// SIMATIC S7-200 project (STEP 7-Micro/WIN), CPU 224XP REL 02.00

SYMBOL_TABLE DR03
S1_0300_AdjDigits0 VW0      // Scale1 - Adjusting digits for zero point
S1_0302_AdjDigits1 VW2      // Scale1 - Adjusting digits for adjusting weight 1
S1_0304_AdjDigits2 VW4      // Scale1 - Adjusting digits for adjusting weight 2
S1_0306_AdjWeight1 VW6      // Scale1 - Adjusting weight 1
S1_0308_AdjWeight2 VW8      // Scale1 - Adjusting weight 2
S1_0310_CharVal  VB10     // Scale1 - Characteristic value [mV/V]
S1_0311_MeasuremTime VB11     // Scale1 - Measurement time, 0=20ms, 1=33,33ms
S1_0312_LimFrequ VB12     // Scale1 - Limit frequency for low pass filter fg
S1_0313_DepthAvValFiltr VB13     // Scale1 - Depth of average value filter [0..255]
S1_0314_ScaleName_maxL VB14     // Scale1 - Scale name, max. length (bytes)
S1_0315_ScaleName_strg VB15     // Scale1 - Scale name, STRING[10]
S1_0326_MinWeight VW26     // Scale1 - Minimum weight for weighing range
S1_0328_MaxWeight VW28     // Scale1 - Maximum weight for weighing range
S1_0330_NumeralStep VW30     // Scale1 - Numeral step (1, 2, 5, 10, 20)
S1_0332_StandstillRange VW32     // Scale1 - Standstill range in weight unit
S1_0334_StandstillTime VD34     // Scale1 - Standstill time in ms
S1_0338_DecimalPoint VB38     // Scale1 - Decimal place for remote display and       ASCII weight output (0...5)
S1_0339_NegZeroRange VB39     // Scale1 - Negative range of zero setting device                   [in % of WBB.]
S1_0340_PosZeroRange VB40     // Scale1 - Positive range of zero setting device                   [in % of WBB.]
S1_0341_TareMax  VB41     // Scale1 - Subtractive tare device range in % of weighing range
S1_0342_TTYinterface VW42     // Scale1 - 0: Siebert S102, 1: ASCII protocol
S1_0344_Res_maxL VB44     // Scale1 - Reserved, max. length (bytes)
S1_0345_Res_strg VB45     // Scale1 - Reserved, STRING[4]
S1_0350_Unit_maxL VB50     // Scale1 - Weight unit for display, max. length (bytes)
S1_0351_Unit_strg VB51     // Scale1 - Weight unit for display, STRING[4]
END_SYMBOL_TABLE

SYMBOL_TABLE DR04
S1_0400_SwOnWeightLim1 VW56     // Scale1 - Switch on point, limit value 1
S1_0402_SwOffWeightLim1 VW58     // Scale1 - Switch off point, limit value 1
S1_0404_SwOnWeightLim2 VW60     // Scale1 - Switch on point, limit value 2
S1_0406_SwOffWeightLim VW62     // Scale1 - Switch off point, limit value 2
S1_0408_LimValParamFlag VB64     // Scale1 - Bit0: 0=lim1 on gross, 1=lim1 on net;                Bit1: --> lim2
S1_0409_Res1     VB65     // Scale1 - Reserve 1
END_SYMBOL_TABLE

SYMBOL_TABLE DR09
S1_0900_ModuleName_maxL VB66     // Scale1 - Name of weighing module, max. length (bytes)
S1_0901_ModuleName_strg VB67     // Scale1 - Name of weighing module, STRING[10]
S1_0912_MLFB_maxL VB78     // Scale1 - MLFB order number, max. length (bytes)
S1_0913_MLFB_strg VB79     // Scale1 - MLFB order number, STRING[20]
S1_0934_Edition1HW VW100    // Scale1 - HW version
S1_0936_FWversion_maxL VB102    // Scale1 - FW version, max. length (bytes)
S1_0937_FWversion_strg VB103    // Scale1 - FW version, STRING[4]
S1_0942_CRCpackage VW108    // Scale1 - Depending on code
END_SYMBOL_TABLE

SYMBOL_TABLE DR15
S1_1500_TareInpVal VW110    // Scale1 - Tare input value (preset Tare pT)
END_SYMBOL_TABLE

SYMBOL_TABLE DR26
S1_2600_Checksum VW112    // Scale1 - Checksum
S1_2602_Res      VB114    // Scale1 - Reserved
S1_2603_PresetTare VB115    // Scale1 - 1 = Tare memory contains ext. default value
S1_2604_Tare_x100 VD116    // Scale1 - Tare weight * 100
S1_2608_ZeroSetVal_x100 VD120    // Scale1 - Zero set value * 100 (set during zero setting)
END_SYMBOL_TABLE

SYMBOL_TABLE DR30
S1_3000_Checksum VW124    // Scale1 - Checksum CRC16
S1_3002_ScaleStatus VW126    // Scale1 - Scale status
S1_3004_OpErrorBits VB128    // Scale1 - Operating error bits
S1_3005_Res1     VB129    // Scale1 - Reserve 1
S1_3006_GrossProcessVal VW130    // Scale1 - Gross weight
S1_3008_NetProcessVal VW132    // Scale1 - Net weight
S1_3010_TareProcessVal VW134    // Scale1 - Tare weight
S1_3012_GNweight VW136    // Scale1 - B/N weight value to display
S1_3014_GNweight10 VD138    // Scale1 - B/N weight value with 10x resolution (basis for ASCII weight value)
S1_3018_TareWeight VW142    // Scale1 - Tare weight value
S1_3020_UnfiltRawVal VW144    // Scale1 - Unfiltered digital value from ADU
S1_3022_FiltRawVal VW146    // Scale1 - Filtered digital value
S1_3024_WghtASCII_maxL VB148    // Scale1 - ASCII weight value, max. length (bytes)
S1_3025_WghtASCII_strg VB149    // Scale1 - ASCII weight value, STRING[14]
S1_3040_Millisecond VW164    // Scale1 - Runtime – Milliseconds (0....999)
S1_3042_Second   VB166    // Scale1 - Runtime – Seconds (0...59)
S1_3043_Minute   VB167    // Scale1 - Runtime – Minutes (0...59)
S1_3044_Hour     VW168    // Scale1 - Runtime – Hours (0...32000)
END_SYMBOL_TABLE

SYMBOL_TABLE MS
Q_S1_Actual_Process_Val VB200    // Scale1 - VBn
Q_S1_Reserve_1   VB201    // Scale1 - VBn+1
Q_S1_Process_Value VW202    // Scale1 - VWn+2
Q_S1_Bit_Messages VB204    // Scale1 - VBn+4
Q_S1_Bit_Messages_Bit0 V204.0   // Scale1 - VBn+4, Bit0, command in progress
Q_S1_Bit_Messages_Bit1 V204.1   // Scale1 - VBn+4, Bit1, command finished ok (TRUE for 1 cycle)
Q_S1_Bit_Messages_Bit2 V204.2   // Scale1 - VBn+4, Bit2, command error (synchronous error) has occurred (TRUE for 1 cycle)
Q_S1_Bit_Messages_Bit3 V204.3   // Scale1 - VBn+4, Bit3, Read/Write-Parameter-Mode is supported
Q_S1_Bit_Messages_Bit4 V204.4   // Scale1 - VBn+4, Bit4, Processvalue not valid!
Q_S1_Bit_Messages_Bit5 V204.5   // Scale1 - VBn+4, Bit5, Reserve
Q_S1_Bit_Messages_Bit6 V204.6   // Scale1 - VBn+4, Bit6, Reserve
Q_S1_Bit_Messages_Bit7 V204.7   // Scale1 - VBn+4, Bit7, Reserve
Q_S1_Sync_Error_Code VB205    // Scale1 - VBn+5
Q_S1_Async_Error_Bits VB206    // Scale1 - VBn+6
Q_S1_Async_Error_Bit0 V206.0   // Scale1 - VBn+6, Bit0, Reboot due to RAM error
Q_S1_Async_Error_Bit1 V206.1   // Scale1 - VBn+6, Bit1, Reboot due to watchdog error
Q_S1_Async_Error_Bit2 V206.2   // Scale1 - VBn+6, Bit2, 24DC power supply faulty/missing
Q_S1_Async_Error_Bit3 V206.3   // Scale1 - VBn+6, Bit3, Number overflow in weight calculation
Q_S1_Async_Error_Bit4 V206.4   // Scale1 - VBn+6, Bit4, Parameter error
Q_S1_Async_Error_Bit5 V206.5   // Scale1 - VBn+6, Bit5, AD converter at limit of measuring range
Q_S1_Async_Error_Bit6 V206.6   // Scale1 - VBn+6, Bit6, Minimum voltage understhot in sensor line
Q_S1_Async_Error_Bit7 V206.7   // Scale1 - VBn+6, Bit7, AD converter fault
Q_S1_Refresh_Counter VB207    // Scale1 - VBn+7
Q_S1_Scale_Status_Bits VW208    // Scale1 - VWn+8
Q_S1_Scale_Status_Bit0 V209.0   // Scale1 - VWn+8, Bit0, Limit value 1 has responded
Q_S1_Scale_Status_Bit1 V209.1   // Scale1 - VWn+8, Bit1, Limit value 2 has responded
Q_S1_Scale_Status_Bit2 V209.2   // Scale1 - VWn+8, Bit2, Tare memory occupied (<>0)
Q_S1_Scale_Status_Bit3 V209.3   // Scale1 - VWn+8, Bit3, Tare memory contains ext. default value
Q_S1_Scale_Status_Bit4 V209.4   // Scale1 - VWn+8, Bit4, Gross weighing range exceeded or understhot (>9 display steps)
Q_S1_Scale_Status_Bit5 V209.5   // Scale1 - VWn+8, Bit5, Gross less than ± 0.25d (d corresponds to set numeral step)
Q_S1_Scale_Status_Bit6 V209.6   // Scale1 - VWn+8, Bit6, Standstill exists
Q_S1_Scale_Status_Bit7 V209.7   // Scale1 - VWn+8, Bit7, Module calibrated
Q_S1_Scale_Status_Bit8 V208.0   // Scale1 - VWn+8, Bit8, Write protect switch active
Q_S1_Scale_Status_Bit9 V208.1   // Scale1 - VWn+8, Bit9, Min. weighing range undershot
Q_S1_Scale_Status_Bit10 V208.2   // Scale1 - VWn+8, Bit10, Reserve
Q_S1_Scale_Status_Bit11 V208.3   // Scale1 - VWn+8, Bit11, Reserve
Q_S1_Scale_Status_Bit12 V208.4   // Scale1 - VWn+8, Bit12, Reserve
Q_S1_Scale_Status_Bit13 V208.5   // Scale1 - VWn+8, Bit13, Reserve
Q_S1_Scale_Status_Bit14 V208.6   // Scale1 - VWn+8, Bit14, startup is running
Q_S1_Scale_Status_Bit15 V208.7   // Scale1 - VWn+8, Bit15, Global module fault / operating error (SF)
Q_S1_Select_Process_Val VB210    // Scale1 - VBn+10
I_S1_Command_Code VB211    // Scale1 - VBn+11
I_S1_Command_Bits VB212    // Scale1 - VBn+12
Q_S1_Reserve_2   VB213    // Scale1 - VBn+13
I_S1_Preset_Tare_Value VW214    // Scale1 - VWn+14
Q_S1_Lifebit_Counter VW216    // Scale1 - VWn+16
Q_S1_Lib_Error_Bits VW218    // Scale1 - VWn+18
Q_S1_RW_Mode_DS_Nr VB220    // Scale1 - VBn+20
Q_S1_RW_Mode_Byte_Offse VB221    // Scale1 - VBn+21
Q_S1_RW_Mode_Write_Data VW222    // Scale1 - VWn+22
Q_S1_RW_Mode_Read_Data VW224    // Scale1 - VWn+24
END_SYMBOL_TABLE

SYMBOL_TABLE User
Error_MS_add     VW298    // Error word of SBR "MicroScale_additional"
Error_Messages1  VW300    // To be displayed at the TP
Error_Messages2  VW302    // To be displayed at the TP
Error_Messages3  VW304    // To be displayed at the TP
Messages_Erase   V306.0   // Button on TP
Command_Trigger  V260.0
Busy             V260.1
Done             V260.2
Aborted          V260.3
Command_Code     VB261
DR               VB262
Offset           VB263
Length           VB264
END_SYMBOL_TABLE

SYMBOL_TABLE MS_add
_S1_Command_Code VB170    // Scale1 - VBn+11
_S1_Word_LoopCounter VB171
_S1_Offset       VB172
_S1_Bit_Messages VB173    // Scale1 - Bit-Messages (Siwarex => PLC)
_S1_Command_INPR V173.0   // Scale1 - command in progress
_S1_Command_FOK  V173.1   // Scale1 - command finished ok
_S1_Command_ERR  V173.2   // Scale1 - command error has occurred
_S1_DR_supported V173.3   // Scale1 - SIWAREX Module supports data record transfer
_S1_Result_bits  VB174
_S1_Busy         V174.0   // Scale1 - identic to OUT parameter
_S1_Done         V174.1
_S1_Aborted      V174.2
_S1_Bytetransfer V174.3
_S1_Err          V174.4
_S1_SequStates   VW175    // Scale1 - Sequencer states
_S1_SequState_08 V176.0   // Scale1 - Waiting for Command_FOK/_ERR of cmd 205
_S1_SequState_09 V176.1   // Scale1 - not used
_S1_SequState_10 V176.2   // Scale1 - Waiting for Actual_Process_Value = prev. Value
_S1_SequState_11 V176.3   // Scale1 - Waiting for next cycle
_S1_SequState_12 V176.4   // Scale1 - Waiting for Actual_Process_Value = 7
_S1_SequState_13 V176.5
_S1_SequState_14 V176.6
_S1_SequState_15 V176.7
_S1_SequState_00 V175.0   // Scale1 - not used
_S1_SequState_01 V175.1   // Scale1 - Waiting for Actual_Process_Value = 7
_S1_SequState_02 V175.2   // Scale1 - No need to wait for Actual_Process_Value valid
_S1_SequState_03 V175.3   // Scale1 - Ready to enter command and trigger start transfer
_S1_SequState_04 V175.4   // Scale1 - Waiting for Command_FOK or Command_ERR
_S1_SequState_05 V175.5   // Scale1 - Read/write finished without error
_S1_SequState_06 V175.6   // Scale1 - Read/write finished with error
_S1_SequState_07 V175.7   // Scale1 - Waiting for Actual_Process_Value = prev. Value
_S1_POINTER      VD177    // Scale1 - Byte address in CPU for read/write job (as pointer)
_S1_Error        VW181
_S1_Prev_Selection VB183
_S1_PackageSize  VB184    // Scale1 - How many words...  (start value)
_S1_PackageCounter VB185    // Scale1 - How many words till transfer interrupt
END_SYMBOL_TABLE

ORGANIZATION_BLOCK MAIN:OB1
TITLE=PROGRAMMKOMMENTARE
VAR
aux1_BOOL:BOOL;	// L0.0 
END_VAR
BEGIN
Network 1 // Call MicroScale
// Netzwerkkommentar
// (network saved uncompiled; FBD cells follow)
// row 0: c1 [MicroScale_V20 ]
// row 1: c1 [ EN:=SM0.0, First_AEW:=AIW4, Second_AEW:=AIW6, Third_AEW:=AIW8, Fourth_AEW:=AIW10, FirstVB_POINTER:=&Q_S1_Actual_Process_Val:VB200, Lib_Error_Bits:=Q_S1_Lib_Error_Bits:VW218, First_AAW=>AQW4, Second_AAW=>AQW6, Third_AAW=>AQW8, Fourth_AAW=>AQW10]
// row 2: c1 [box]
// row 3: c1 [box]
// row 4: c1 [box]
// row 5: c1 [box]
// row 6: c1 [box]
// row 7: c1 [box]
Network 2 // Call MicroScale_additional
LD     SM0.0
CALL   MicroScale_additional:SBR0, &Q_S1_Actual_Process_Val:VB200, &VB0, Command_Code:VB261, DR:VB262, Offset:VB263, Length:VB264, Command_Trigger:V260.0, Busy:V260.1, Done:V260.2, Aborted:V260.3, Error_MS_add:VW298
Network 3 // Create pulse of "Aborted"
LD     Aborted:V260.3
EU
=      #aux1_BOOL:L0.0
Network 4
LD     SM0.0
CALL   TP177micro:SBR3, VB218, Q_S1_Async_Error_Bits:VB206, Q_S1_Sync_Error_Code:VB205, Error_MS_add:VW298, #aux1_BOOL:L0.0, Error_Messages1:VW300, Error_Messages2:VW302, Error_Messages3:VW304, Messages_Erase:V306.0
END_ORGANIZATION_BLOCK

// SBR0: protected block, not included

// SBR1: protected block, not included

SUBROUTINE_BLOCK TP177micro:SBR3
TITLE=UNTERPROGRAMM-KOMMENTARE
VAR_INPUT
Lib_Error_Bits:BYTE;	// LB0  Library_Error_Bits
Asyn_Error_Bits:BYTE;	// LB1  Asynchronous Error Bits
Syn_Error_Code:BYTE;	// LB2  Synchronous Error Code
Error_MS_add:INT;	// LW3  MicroScale_additional errors
Trigger_pulse:BOOL;	// L5.0  Pulse for 1 cycle
END_VAR
VAR_IN_OUT
Error_Messages1:WORD;	// LW6  Error messages for Panel
Error_Messages2:WORD;	// LW8  Error messages for Panel
Error_Messages3:WORD;	// LW10  Error messages for Panel
Messages_Erase:BOOL;	// L12.0  Error messages erase for Panel
END_VAR
BEGIN
Network 1 //  Netzwerktitel
//  Netzwerkkommentar
// (network saved uncompiled; FBD cells follow)
// row 0: c4 [MOV_W ]
// row 1: c1 [AND #Messages_Erase:L12.0 ]  c2 -- v  c3 --  c4 [ EN:=power@row1, IN:=0, ENO=>V?0, OUT=>#Error_Messages1:LW6]
// row 2: c2 ^v  c4 [box]
// row 3: c2 ^v  c4 [MOV_W ]
// row 4: c2 ^v  c3 --  c4 [ EN:=power@row4, IN:=0, ENO=>V?0, OUT=>#Error_Messages2:LW8]
// row 5: c2 ^v  c4 [box]
// row 6: c2 ^v  c4 [MOV_W ]
// row 7: c2 ^v  c3 --  c4 [ EN:=power@row7, IN:=0, ENO=>V?0, OUT=>#Error_Messages3:LW10]
// row 8: c2 ^v  c4 [box]
// row 9: c2 ^v
// row 10: c2 ^  c3 --  c4 [R #Messages_Erase:L12.0 N:=1]
// row 11: c4 [box]
Network 2
LD     SM0.1
R      L7.2, 1
Network 3
//The ORB instruction ORs the corresponding bits of two input values
// (network saved uncompiled; FBD cells follow)
// row 0: c4 [WOR_B ]
// row 1: c1 [AND SM0.0 ]  c2 -- v  c3 --  c4 [ EN:=power@row1, IN1:=#Lib_Error_Bits:LB0, IN2:=LB6, ENO=>V?0, OUT=>LB6]
// row 2: c2 ^v  c4 [box]
// row 3: c2 ^v  c4 [box]
// row 4: c2 ^v  c4 [WOR_B ]
// row 5: c2 ^  c3 --  c4 [ EN:=power@row5, IN1:=#Asyn_Error_Bits:LB1, IN2:=LB7, ENO=>V?0, OUT=>LB7]
// row 6: c4 [box]
// row 7: c4 [box]
Network 4
LDN    #Trigger_pulse:L5.0
JMP    10
Network 5
LDB=   #Syn_Error_Code:LB2, 1
S      L9.0, 1
Network 6
LDB=   #Syn_Error_Code:LB2, 2
S      L9.1, 1
Network 7
LDB=   #Syn_Error_Code:LB2, 4
S      L9.2, 1
Network 8
LDB=   #Syn_Error_Code:LB2, 5
S      L9.3, 1
Network 9
LDB=   #Syn_Error_Code:LB2, 7
S      L9.4, 1
Network 10
LDB=   #Syn_Error_Code:LB2, 8
S      L9.5, 1
Network 11
LDB=   #Syn_Error_Code:LB2, 20
S      L9.6, 1
Network 12
LDB=   #Syn_Error_Code:LB2, 21
S      L9.7, 1
Network 13
LDB=   #Syn_Error_Code:LB2, 77
S      L8.0, 1
Network 14
LDB=   #Syn_Error_Code:LB2, 80
S      L8.2, 1
Network 15
LDB=   #Syn_Error_Code:LB2, 81
S      L8.3, 1
Network 16
LDB=   #Syn_Error_Code:LB2, 82
S      L8.4, 1
Network 17
LDB=   #Syn_Error_Code:LB2, 83
S      L8.5, 1
Network 18
LDB=   #Syn_Error_Code:LB2, 84
S      L8.6, 1
Network 19
LDB=   #Syn_Error_Code:LB2, 85
S      L8.7, 1
Network 20
LDB=   #Syn_Error_Code:LB2, 86
S      L11.0, 1
Network 21
LDB=   #Syn_Error_Code:LB2, 87
S      L11.1, 1
Network 22
LDB=   #Syn_Error_Code:LB2, 88
S      L11.2, 1
Network 23
LDB=   #Syn_Error_Code:LB2, 94
S      L11.3, 1
Network 24
LDB=   #Syn_Error_Code:LB2, 96
S      L11.4, 1
Network 25
LDB=   #Syn_Error_Code:LB2, 100
S      L11.5, 1
Network 26
LDB=   #Syn_Error_Code:LB2, 171
S      L11.6, 1
Network 27
LDB=   #Syn_Error_Code:LB2, 172
S      L11.7, 1
Network 28
LDB=   #Syn_Error_Code:LB2, 173
S      L10.0, 1
Network 29
LDW=   #Error_MS_add:LW3, 1
S      L10.3, 1
Network 30
LDW=   #Error_MS_add:LW3, 2
S      L10.4, 1
Network 31
LDW=   #Error_MS_add:LW3, 3
S      L10.5, 1
Network 32
LDW=   #Error_MS_add:LW3, 4
S      L10.6, 1
Network 33
LBL    10
END_SUBROUTINE_BLOCK

DATA_BLOCK_TAB DataRecords
BEGIN
//DR3
         S1_0300_AdjDigits0, 5461
         S1_0302_AdjDigits1, 60074
         S1_0304_AdjDigits2, 0
         S1_0306_AdjWeight1, 2000
         S1_0308_AdjWeight2, 0
         S1_0310_CharVal, 2
         S1_0311_MeasuremTime, 0
         S1_0312_LimFrequ, 4
         S1_0313_DepthAvValFiltr, 15
         S1_0314_ScaleName_maxL, 10
         S1_0315_ScaleName_strg, "SIWAREX MS"
         S1_0326_MinWeight, 20
         S1_0328_MaxWeight, 2000
         S1_0330_NumeralStep, 1
         S1_0332_StandstillRange, 10
         S1_0334_StandstillTime, 1000
         S1_0338_DecimalPoint, 2
         S1_0339_NegZeroRange, 10
         S1_0340_PosZeroRange, 10
         S1_0341_TareMax, 100
         S1_0342_TTYinterface, 0
         S1_0344_Res_maxL, 4
         S1_0345_Res_strg, "----"
         S1_0350_Unit_maxL, 4
         S1_0351_Unit_strg, " kg "
//DR4
         S1_0400_SwOnWeightLim1, 400
         S1_0402_SwOffWeightLim1, 220
         S1_0404_SwOnWeightLim2, 1000
         S1_0406_SwOffWeightLim, 980
         S1_0408_LimValParamFlag, 2#0
         S1_0409_Res1, 0
//DR9
         S1_0900_ModuleName_maxL, 10
         S1_0901_ModuleName_strg, "SIWAREX MS"
         S1_0912_MLFB_maxL, 20
         S1_0913_MLFB_strg, "7MH4930-0AA01       "
         S1_0934_Edition1HW, 1
         S1_0936_FWversion_maxL, 4
         S1_0937_FWversion_strg, "F1.3"
         S1_0942_CRCpackage, 16817
//DR15
         S1_1500_TareInpVal, 0
//DR26
         S1_2600_Checksum, 26097
         S1_2602_Res, 0
         S1_2603_PresetTare, 0
         S1_2604_Tare_x100, 0
         S1_2608_ZeroSetVal_x100, 0
//DR30
         S1_3000_Checksum, 405
         S1_3002_ScaleStatus, 2#11000000
         S1_3004_OpErrorBits, 0
         S1_3005_Res1, 0
         S1_3006_GrossProcessVal, 60
         S1_3008_NetProcessVal, 60
         S1_3010_TareProcessVal, 0
         S1_3012_GNweight, 60
         S1_3014_GNweight10, 604
         S1_3018_TareWeight, 0
         S1_3020_UnfiltRawVal, 7110
         S1_3022_FiltRawVal, 7110
         S1_3024_WghtASCII_maxL, 14
         S1_3025_WghtASCII_strg, "      0,60 kg "
         S1_3040_Millisecond, 280
         S1_3042_Second, 18
         S1_3043_Minute, 45
         S1_3044_Hour, 0
END_DATA_BLOCK_TAB
